(* PLC project Sin nombre, Desconocido Sin nombre 1 *)
(* stored: creationDateTime 2022-10-17T16:56:25, modificationDateTime 2023-09-28T08:07:46 *)

PROGRAM program0
  VAR
    sensor AT %IX0.0 : BOOL := 0;
    led_sensor AT %QX0.2 : BOOL := 0;
    led_red AT %QX0.1 : BOOL := 0;
    led_green AT %QX0.0 : BOOL := 0;
    relay AT %QX0.3 : BOOL := 0;
  END_VAR
  VAR
    temporizador : TIME := T#10000ms;
    tiempo_sensor : TIME := T#500ms;
    TOF1 : TOF;
    TP1 : TP;
  END_VAR
  VAR  (* added by the conversion: wires and edge detectors of the diagram *)
    _NOT26_OUT : BOOL;
  END_VAR

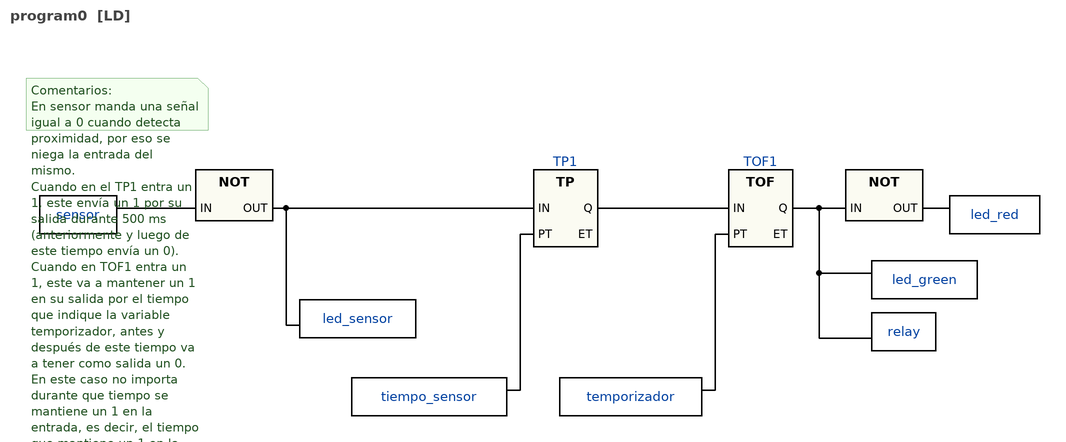
(* LD diagram, written out as Structured Text *)
(* Comentarios:
En sensor manda una señal igual a 0 cuando detecta proximidad, por eso se niega la entrada del mismo. 
Cuando en el TP1 entra un 1, este envía un 1 por su salida durante 500 ms (anteriormente y luego de este tiempo envía un 0).
Cuando en TOF1 entra un 1, este va a mantener un 1 en su salida por el tiempo que indique la variable temporizador, antes y después de este tiempo va a tener como salida un 0. En este caso no importa durante que tiempo se mantiene un 1 en la entrada, es decir, el tiempo que mantiene un 1 en la salida es independiente de cuanto dura el 1 en la entrada.
Según la salida de TOF1 se activará el relay junto con el led_green o el led_red, o todo lo contario.
En cuanto al led_sensor, este se activa cada vez que el sensor detecta proximidad y se paga en caso contrario. *)
_NOT26_OUT := NOT sensor;
TP1(IN := _NOT26_OUT, PT := tiempo_sensor);
TOF1(IN := TP1.Q, PT := temporizador);
led_red := NOT TOF1.Q;
led_green := TOF1.Q;
led_sensor := _NOT26_OUT;
relay := TOF1.Q;
END_PROGRAM

CONFIGURATION Config0
  RESOURCE Res0 ON PLC
    TASK task0(INTERVAL := T#20ms, PRIORITY := 0);
    PROGRAM instance0 WITH task0 : program0;
  END_RESOURCE
END_CONFIGURATION
